Staubli VAL3: checkPCircle.pgx

public program checkPCircle(num x_nIndex, point x_pToCheck, num& x_nResult[])
  local num i
  local bool l_bDistance[3]
  local bool l_bUnreach
  local frame l_fFrame
  local num l_nDistance
  local num l_nNewDist
  local num l_nStep
  local num l_nTo
  local point l_pCircle[3]
  local point l_pPoint
  local tool l_tTool
begin
  // check if the x_pToCheck is inside the Circle
  //
  //  INIT
  //
  l_nDistance=1000
  l_nStep=x_nResult=-1
  call tcp:getTool(l_tTool,pEditPoint.nIndexTool)
  l_pPoint=here(l_tTool,pEditPoint.fFrame)
  // get the three point
  if x_nIndex>0
    call getPoint(l_pCircle,false,x_nIndex-1)
    call getPoint(l_pCircle[1],false,x_nIndex)
  endIf
  // check if the points are the same
  l_bDistance=distance(position(l_pCircle,pEditPoint.fFrame),position(l_pCircle[2],pEditPoint.fFrame))<1
  l_bDistance[1]=distance(position(l_pCircle[1],pEditPoint.fFrame),position(l_pCircle[2],pEditPoint.fFrame))<1
  l_bDistance[2]=distance(position(l_pCircle,pEditPoint.fFrame),position(l_pCircle[1],pEditPoint.fFrame))<1
  call isReachable(l_pCircle,l_tTool,l_bUnreach)
  if !l_bUnreach
    call isReachable(l_pCircle[1],l_tTool,l_bUnreach)
    // check the frame
    if !l_bUnreach
      l_bUnreach=setFrame(l_pCircle,l_pCircle[2],l_pCircle[1],fSetFrame)!=0
    endIf
  endIf
  if l_bDistance or l_bDistance[1] or l_bDistance[2] or l_bUnreach
    // not valid circle point
    x_nResult=-1
    return
  endIf
  // first check step 0.1
  for i=0 to 1 step 0.1
    l_pPoint.trsf=interpolateC(position(l_pCircle,pEditPoint.fFrame),position(l_pCircle[2],pEditPoint.fFrame),position(l_pCircle[1],pEditPoint.fFrame),i)
    l_nNewDist=distance(x_pToCheck.trsf,l_pPoint.trsf)
    if l_nNewDist<l_nDistance
      l_nDistance=l_nNewDist
      l_nStep=i
    endIf
  endFor
  if l_nStep!=-1
    // second step 0.01
    l_nTo=min(l_nStep+0.05,1)
    for i=max(l_nStep-0.05,0) to l_nTo step 0.01
      l_pPoint.trsf=interpolateC(position(l_pCircle,pEditPoint.fFrame),position(l_pCircle[2],pEditPoint.fFrame),position(l_pCircle[1],pEditPoint.fFrame),i)
      l_nNewDist=distance(x_pToCheck.trsf,l_pPoint.trsf)
      if l_nNewDist<l_nDistance
        l_nDistance=l_nNewDist
        l_nStep=i
      endIf
    endFor
  endIf
  if l_nStep!=-1
    // third step 0.001
    l_nTo=min(l_nStep+0.005,1)
    for i=max(l_nStep-0.005,0) to l_nTo step 0.001
      l_pPoint.trsf=interpolateC(position(l_pCircle,pEditPoint.fFrame),position(l_pCircle[2],pEditPoint.fFrame),position(l_pCircle[1],pEditPoint.fFrame),i)
      l_nNewDist=distance(x_pToCheck.trsf,l_pPoint.trsf)
      if l_nNewDist<l_nDistance
        l_nDistance=l_nNewDist
        l_nStep=i
      endIf
    endFor
  endIf
  // 5 mm tollerance
  if l_nDistance<=5
    // store the value
    x_nResult=l_nStep
  endIf
end
